TYPE typeNewMsgHeader :
STRUCT
	
col1:STRING :='Time Raised';
col2:STRING :='Time Resolved';
col3:STRING :='Message Text';
col4:STRING :='Message Location';
col5:STRING :='test1';





END_STRUCT
END_TYPE

(* stored: Version 1.1.0.1, ProductVersion 3.1.4024.12
   DUT typeNewMsgHeader: Id {caecb989-aec8-4d1a-b4f1-2919b401fa30} *)
